FUNCTION_BLOCK FB_SimulateProcess IMPLEMENTS I_StationProcess
VAR
	_ProcessTime	: TIME;
END_VAR

METHOD Execute : BOOL
VAR_INPUT
	Mover	: XPlanarApplication.I_XPlanarMover;
END_VAR

VAR_INST
	SimulateTimer: TON;
END_VAR
SimulateTimer(IN := Mover <> 0, PT := _ProcessTime);
IF SimulateTimer.Q THEN
	SimulateTimer(IN := FALSE);
	Execute := TRUE; //Set Execute to TRUE when process is complete and station base will send mover to next station.
END_IF
END_METHOD

PROPERTY ProcessTime : LREAL
SET
_ProcessTime := TO_TIME(ProcessTime * 1000);
END_SET
END_PROPERTY

END_FUNCTION_BLOCK

(* stored: Version 1.1.0.1
   POU FB_SimulateProcess: Id {e15be128-38cd-4b88-b277-99cc8805ba93}, SpecialFunc None
   Method Execute: Id {55077361-cf1d-469f-9e7d-1a06c60a682a}
   Property ProcessTime: Id {88016f18-daea-4c24-9e42-8f2f427351e2}
   Set Set: Id {0ab05e10-a647-4e4f-9f04-f5905abf574e} *)
